FUNCTION_BLOCK FB_Blinken_Ampel
VAR_INPUT
	tPeriode  : TIME := T#1S;   // Gesamtperiode des Blinkens
END_VAR
VAR_OUTPUT
	bBlink : BOOL := FALSE;     // Ausgang: Blinkt true/false
END_VAR
VAR
	fbTon : TON;                // Einschalt-Timer
END_VAR

// Timer läuft dauerhaft
fbTon(IN := TRUE, PT := tPeriode);

// Blink-Logik: 50/50 Duty Cycle
IF fbTon.ET < tPeriode / 2 THEN
	bBlink := TRUE;
ELSE
	bBlink := FALSE;
END_IF

// Timer neu starten, wenn abgelaufen
IF fbTon.Q THEN
	fbTon(IN := FALSE);  // kurzer Reset
END_IF

END_FUNCTION_BLOCK

(* stored: Version 1.1.0.1, ProductVersion 3.1.4024.15
   POU FB_Blinken_Ampel: Id {7c371093-a381-4e7c-928f-e6a4df91eda3}, SpecialFunc None *)
